// TwinCAT 3 PLC project test
// ProgramVersion: 3.1.4023.0
// CompilerDefines: VISU_USEWSTRING
// libraries:
//   Tc2_MC2, * (Beckhoff Automation GmbH)
//   Tc2_Standard, * (Beckhoff Automation GmbH)
//   Tc2_System, * (Beckhoff Automation GmbH)
//   Tc3_Module, * (Beckhoff Automation GmbH)
//   VisuDialogs, * (System)
//   VisuSymbols,3.5.10.0,System
// project tree:
//   / GlobalTextList.TcGTLO, PlcTask.TcTTO, VisualizationManager.TcVMO (not stored), VISU_TASK.TcTTO
//   POUs/ MAIN.TcPOU
//   POUs/single/ single.TcPOU
//   VISUs/ singleAxis.TcVIS
// real-time tasks:
//   TASK PlcTask: cycle T#10ms, priority 20, ADS port 350
//   TASK VISU_TASK: cycle T#200000us, priority 30, ADS port 351
// motion (NC):
//   TASK NC-Task 1 SAF: cycle T#2ms, priority 4, ADS port 501
//   TASK NC-Task 1 SVB: cycle T#10ms, priority 8, ADS port 511
//   AXIS Axis 1 (id 1)
//     Dynamic: Acceleration=50, Deceleration=50
//     Velo: SlowManual=50, FastManual=200
//     OtherSettings: AllowMotionCmdToSlave=true
//     encoder EncType=19
//       EncPara: ScaleFactorNumerator=5, ScaleFactorDenominator=524288, MaxCount=#xffffffff
//     drive DrvType=16
//       DrvPara: MaxCount=#xffffffff, DriveControlDWord=#x00020000
//         Analog: TorqueSetpointScale=10, ScaleFactorActTorque=0.1
//         TimeComp: TaskDelayCycles=1
//     controller CtrType=1
//       CtrPara: PriorControlFactor=1
//         PosDiffControl: Range=5000
//         Observer: BandWidth=20
// I/O:
//   DEVICE Device 3 (EtherCAT), AmsNetId 169.254.203.149.4.1
//     Drive 1 (L7N - Standard EtherCAT drive) [L7N - Standard EtherCAT drive(CoE)]
// variable links:
//   NC-Task 1 SAF/Axes/Axis 1 <-> Device 3 (EtherCAT)/Drive 1 (L7N - Standard EtherCAT drive)
//     Drive/Inputs/In/nDcOutputTime <-> InfoData/DcOutputShift
//     Drive/Inputs/In/nState1 <-> 2nd Transmit PDO mapping/Statusword
//     Drive/Inputs/In/nState2 <-> 2nd Transmit PDO mapping/Statusword @bit 8
//     Drive/Inputs/In/nState4 @bit 1 <-> WcState/InputToggle
//     Drive/Inputs/In/nState4 <-> WcState/WcStateIn
//     Drive/Outputs/Out/nCtrl1 <-> 2nd Receive PDO mapping/Controlword
//     Drive/Outputs/Out/nCtrl2 <-> 2nd Receive PDO mapping/Controlword @bit 8
//     Drive/Outputs/Out/nDataOut1 <-> 2nd Receive PDO mapping/Target Position
//     Enc/Inputs/In/nDataIn1 <-> 2nd Transmit PDO mapping/Position Actual Value
//     Enc/Inputs/In/nDcInputTime <-> InfoData/DcInputShift
//     Enc/Inputs/In/nState4 @bit 1 <-> WcState/InputToggle
//     Enc/Inputs/In/nState4 <-> WcState/WcStateIn
//   test/test Instance <-> NC-Task 1 SAF/Axes/Axis 1
//     PlcTask Inputs/single.axisx.NcToPlc <-> Outputs/ToPlc
//     PlcTask Outputs/single.axisx.PlcToNc <-> Inputs/FromPlc

CONFIGURATION test
    RESOURCE PLC ON TwinCAT3
        TASK PlcTask(INTERVAL := T#10ms, PRIORITY := 20);
        TASK VISU_TASK(INTERVAL := T#200000us, PRIORITY := 30);
        PROGRAM MAIN WITH PlcTask : MAIN;
        PROGRAM VisuElems_Visu_Prg WITH VISU_TASK : VisuElems.Visu_Prg;
    END_RESOURCE
END_CONFIGURATION

// ---- POUs/MAIN.TcPOU
PROGRAM MAIN
VAR

END_VAR

single.checkPower();
single.checkMoving();
single.checkRelMove();
single.checkHalt();
single.checkStop();
single.checkReset();
single.checkAdjustingVelocity();
single.checkSetPoint();
single.checkGoHome();

END_PROGRAM

// ---- POUs/single/single.TcPOU
PROGRAM single
VAR
	axisx: AXIS_REF;

	mcPower: MC_Power;
	shouldPowerOn: BOOL;
	isMotorReady: BOOL;
	
	mcSetPosition: MC_SetPosition;
	shouldSetZero: BOOL;
	
	mcJog: MC_Jog;
	shouldJog: BOOL;
	jogDirection: BOOL;
	
	mcMoveRelative: MC_MoveRelative;
	shouldMoveRel: BOOL;
	
	mcHalt: MC_Halt;
	shouldHalt: BOOL;
	
	mcStop: MC_Stop;
	shouldStop:BOOL;
	
	mcReset: MC_Reset;
	shouldReset: BOOL;
	
	mcMoveVelocity: MC_MoveVelocity;
	shouldAdjustVelocity: BOOL;
	velocity: INT;
	
	mcHome: MC_Home;
	shouldGoHome: BOOL;
	homeTrigger: BOOL;
END_VAR

METHOD checkAdjustingVelocity : BOOL
VAR
END_VAR
IF isMotorReady THEN
	mcMoveVelocity(
		Axis:= axisx, 
		Execute:= shouldAdjustVelocity,
		Velocity:= velocity );
END_IF
END_METHOD

METHOD checkGoHome : BOOL
VAR_INPUT
END_VAR
mcHome(
	Axis:= axisx, 
	Execute:= shouldGoHome, 
	Position:= 0, 
	bCalibrationCam:= homeTrigger
);
END_METHOD

METHOD checkHalt : BOOL
VAR_INPUT
END_VAR
IF isMotorReady THEN
	mcHalt(
		Axis:= axisx, 
		Execute:= shouldHalt);
END_IF
END_METHOD

METHOD checkMoving : BOOL
VAR_STAT
END_VAR
IF isMotorReady THEN
	IF shouldJog THEN
		IF jogDirection THEN
		mcJog(
			Axis:= axisx, 
			JogForward:= TRUE, 
			JogBackwards:= FALSE,
			Velocity:= 50);
		ELSE
			mcJog(
				Axis:= axisx, 
				JogForward:= FALSE, 
				JogBackwards:= TRUE,
				Velocity:= 50);
		END_IF
	END_IF
END_IF
END_METHOD

METHOD checkPower : BOOL
VAR_INPUT
END_VAR
VAR
END_VAR
mcPower(
	Axis:= axisx, 
	Enable:= shouldPowerOn, 
	Enable_Positive:= TRUE, 
	Enable_Negative:= TRUE,
	Status=> isMotorReady);
END_METHOD

METHOD checkRelMove : BOOL
VAR_STAT
END_VAR
IF isMotorReady THEN
	mcMoveRelative(
		Axis:= axisx, 
		Execute:= shouldMoveRel, 
		Distance:= 2000, 
		Velocity:= 50);
END_IF;
END_METHOD

METHOD checkReset : BOOL
IF isMotorReady THEN
	mcReset(
		Axis:= axisx, 
		Execute:= shouldReset);
END_IF
END_METHOD

ACTION checkSetPoint:
mcSetPosition(
	Axis:= axisx, 
	Execute:= shouldSetZero,
	Position := 0);
END_ACTION

METHOD checkStop : BOOL
VAR

END_VAR
IF isMotorReady THEN
	mcStop(
		Axis:= axisx, 
		Execute:= shouldStop);
END_IF
END_METHOD

END_PROGRAM

// ---- GlobalTextList.TcGTLO
TEXTLIST GlobalTextList
  102 = '%.2f'
  174 = '%d'
  303 = 'direction'
  92 = 'halt'
  340 = 'jog'
  920 = 'move'
  232 = 'power'
  793 = 'relative move'
  341 = 'reset'
  944 = 'set position'
  838 = 'stop'
  297 = 'stop1'
  201 = 'stop_execute_false'
  580 = 'timer'
  366 = '上电'
  163 = '停机'
  859 = '停止'
  882 = '动态耦合'
  567 = '反转'
  183 = '开机'
  357 = '循环转'
  798 = '断电'
  959 = '方向'
  315 = '正传'
  27 = '正反转'
  647 = '正转'
  147 = '电源'
  754 = '相对位置移动'
  217 = '设置原点'
  628 = '调速'
  891 = '转动'
  781 = '静态耦合'
  383 = '静态解耦'
END_TEXTLIST

// ---- VISUs/singleAxis.TcVIS
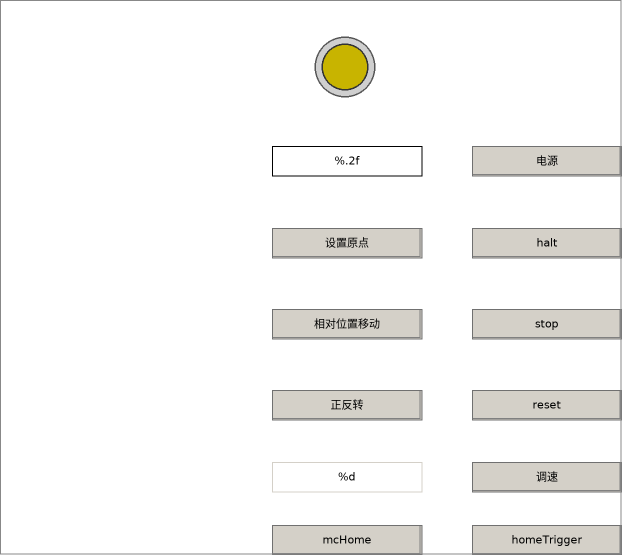
VISUALIZATION singleAxis  // 622x555
    Rectangle (272,146 150x30), "%.2f", text variable: single.axisx.NcToPlc.ActPos
    Button (272,390 150x30), "正反转"
        OnMouseClick: toggle single.jogDirection
        OnMouseClick: execute { single.shouldJog := TRUE; }
    Lamp1 (310,32 70x70), variable: single.axisx.NcToPlc.StateDWord.20, style: Lamp-Lamp1-Yellow
    Button (272,309 150x30), "相对位置移动"
        tap single.shouldMoveRel
    Button (272,228 150x30), "设置原点"
        tap single.shouldSetZero
    Button (472,146 150x30), "电源"
        toggle single.shouldPowerOn
    Button (472,228 150x30), "halt"
        tap single.shouldHalt
    Button (472,309 150x30), "stop"
        tap single.shouldStop
    Button (472,462 150x30), "调速"
        tap single.shouldAdjustVelocity
    Textfield (272,462 150x30), "%d", text variable: single.velocity
        OnMouseClick: write single.velocity via VisuDialogs.Numpad, min 10, max 500
    Button (472,390 150x30), "reset"
        tap single.shouldReset
    Button (272,525 150x30), "mcHome"
        tap single.shouldGoHome
    Button (472,525 150x30), "homeTrigger"
        tap single.homeTrigger
END_VISUALIZATION
